{attribute 'global_init_slot' := '49991'}
{attribute 'qualified_only'}
VAR_GLOBAL CONSTANT
	(* cart joints are defiend in sequence as below
	[monitor lift, monitor rotate, armset, pedal] *)
	
	// encoder resolution
	g_incEncoderRes :ARRAY[1..4] OF DINT :=[4(65536)];
	g_absEncoderRes :ARRAY[1..4] OF DINT :=[16777216,131072,16777216,16777216];
	
	// reduction ratio
	g_motorReduction :ARRAY[1..4] OF LREAL :=[2*pi/0.0004682,3317.76,2*pi/0.0004682,1.5*138.0/5*2*pi/0.004];
	// TODO: need to be verified, especially joint2
	g_absEncoderReduction :ARRAY[1..4] OF LREAL :=[1.534, 1 , 1.534, 1.534];// 2*pi/(reduction*g_absEncoderRes)=Line_Resolution_car(from old code, 0.001*2/2^13)
	
	// motor parameters
	g_motorTrqConst :ARRAY[1..4] OF LREAL :=[4(0.0292)];
	g_motorMaxCurrent :ARRAY[1..4] OF LREAL :=[4(1000)];//mA
	
	// motor and absEncoder direction
	g_motorDir :ARRAY[1..4] OF INT :=[1, -1, 1, 1];
	g_asbEncoderDir :ARRAY[1..4] OF INT :=[-1, -1, -1, 1];
																 
	// joint position limit
	g_minJntPos: ARRAY[1..4] OF LREAL:=[0,-(56.24901883)*g_deg2Rad,0,0];
	g_maxJntPos: ARRAY[1..4] OF LREAL:=[0.40,-(21.7523482+2)*g_deg2Rad,0.30,0.20];
	
	// joint motion velocity 
	g_jntCtrlMotionVel :ARRAY[1..7] OF LREAL :=[0.015,2*g_deg2Rad,0.01,0.0075]; //0.0075
	g_jntCtrlMotionAcc :ARRAY[1..7] OF LREAL :=[0.015*2,2*2*g_deg2Rad,0.01*2,0.0075*2]; //0.0075
	
	g_jntVelMax : ARRAY[1..4] OF LREAL := [0.015,2*g_deg2Rad,0.01,0.0075];
	//cart monitor angle parameter
	g_monitorAnglePara : ST_MonitorAnglePara;
END_VAR

(* stored: Version 1.1.0.1, ProductVersion 3.1.4024.11
   GVL GVL_CartJointParameters: Id {c84079e2-419b-45d5-aeb0-1f4f362f3cde} *)
